(*
Nazwa:			P01_BottleFeeder
Opis:			Stacja podajnika nasadek
Wersja:			v0.1
Data:			2018-10-10
Autor:			DP
Urzadzenia:		
Konfiguracja:	
Info:

*)
PROGRAM P01_BottleFeeder
VAR_INPUT
	IbBottleFeederGate1Sensor					:BOOL;			// Czujnik otwarcia 1 szlabanu 
	IbBottleFeederGate2Sensor					:BOOL;			// Czujnik otwarcia 2 szlabanu 
	IbBottleFeederArmLeftSensor					:BOOL;			// Czujnik położenia siłownika poziomego ramienia - lewy
	IbBottleFeederArmRightSensor				:BOOL;			// Czujnik położenia siłownika poziomego ramienia - prawy
	IbBottleFeederArmUpSensor					:BOOL;			// Czujnik położenia siłownika pionowego ramienia - góra
	IbBottleFeederArmDownSensor					:BOOL;			// Czujnik polożenia siłowniak pionowego ramienia - dół
	IbBottleFeederFormPositioningClosedSensor	:BOOL;			// Czujnik schowania siłownika pozycjonujacego formatke
	IbBottleFeederBottleSensor					:BOOL;			// Czujnik obecności butelki pomiedzy szlabanami
	IbBottleFeederFormGateBeforeSensor 			:BOOL;			// Czujnik przed szlabanem formatek
	IbBottleFeederFormGateAfterSensor 			:BOOL;			// Czujnik za szlabanem formatek
	IbBottleFeederLevelSensor					:BOOL;			// Czujnik kolejki butelki
	IbBottleFeederNotInsertedSensor				AT %I*: BOOL; 	// Czujnik źle włozonej butelki za stacją	
	
END_VAR

VAR
	tonSimu1	:	TON;
	tonSimu2	:	TON;	
	tonSimu3	:	TON;	

	fbBottleFeeder						  	: FB_BottleFeeder;		// Bloczek do obsługi stacji podajnika butelek
	fbTurnTable								: FB_MitsubishiInverter; 	//Bloczek do obsługi falownika stołu obrotewego
	
	eBottleFeederStationState				: E_Station;
	eBottleFeederRunningState				: E_BottleFeederState;
	fbBottleFeederState						: FB_State;
	
	eBottleFeederTurnTableState				: E_Station;
	eBottleFeederTurnTableRunningState		: E_ConveyorState;
	fbBottleSorterTurnTableState			: FB_State;
	
	fbGateBottleFeeder						: FB_SpringGateV2;
	
	//Wyjścia sterujące
	QbBottleFeederGate1						:BOOL;			// Szlaban 1 (lewy)
	QbBottleFeederGate2						:BOOL;			// Szlaban 2 (prawy)
	QbBottleFeederArmLeft					:BOOL;			// Lewo
	QbBottleFeederArmDown					:BOOL;			// Dół
	QbBottleFeederGripper					:BOOL;			// Chwytak
	QbBottleFeederFormPositioning			:BOOL;			// Pozycjonowanie formatki
	QbBottleFeederFormGate					:BOOL;			// Szlaban formatki
	
	// Stół obrotowy
	uiBottleFeederTurnTableSW					AT %I*: UINT;
	uiBottleFeederTurnTableActualVelocity		AT %I*: UDINT;
	uiBottleFeederTurnTableCW  					AT %Q*: UINT;
	udiBottleFeederTurnTableVelocity			AT %Q*: UDINT;
	bGateRun: BOOL;
	iTest2: INT;
	bTestTurnTableRun: BOOL;
	
	bTest: BOOL;
	tonNotQbBottleFeederArmDown: TON;
END_VAR

aWarning();
aBottleFeeder();
aTurntable();
aGateTime();
aGate();

tonNotQbBottleFeederArmDown(IN:= NOT QbBottleFeederArmDown, PT:=T#50MS);


VIS.nBottleFeederTurnTableVelocityCV := uiBottleFeederTurnTableActualVelocity;

IF fbBottleFeeder.bCycleDone THEN
	bGateRun:=TRUE;
END_IF

IF fbGateBottleFeeder.bCycleDone THEN
	bGateRun:=FALSE;
END_IF

(********ASOWANIE ROZKAZÓW CYKLI*********)
IF fbBottleFeeder.bCycleDone AND bManualMode THEN
	VIS.bBottleFeederRun := FALSE;
END_IF


fbBottleFeederState(
	eState									:= eBottleFeederStationState,
	bRun									:= VIS.bBottleFeederRun,
	eBottleSorterRunningState				:= eBottleFeederRunningState,
	sStateDesc								=> VIS.sBottleFeederState,
	iState									=> VIS.iBottleFeederState);
	
(*
// tutaj dorobić obsługe wizki dla stoli obrotowego
eBottleSorterTurnTableRunningState:=eBottleSorterTurnTableState;


fbBottleSorterTurnTableState(
	eState													:= eBottleSorterTurnTableState , 
	bRun													:= GVL.bBottleSorterTurnTableRun,	
	eBottleSorterRunningState									:= eBottleSorterTurnTableRunningState , 
	sStateDesc												=> VIS.sBottleSorterTurnTableState,
	iState													=> VIS.iBottleSorterTurnTableState	);
*)

ACTION aBottleFeeder:
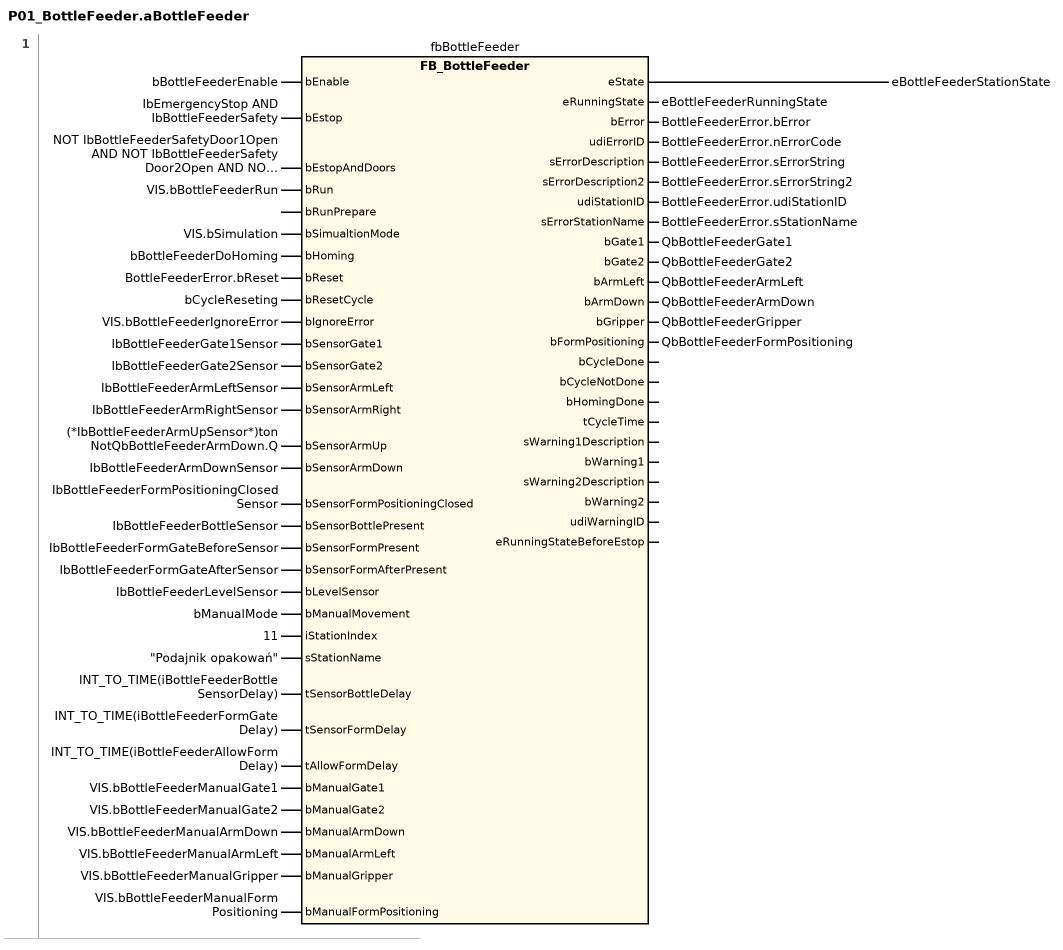
// NETWORK 1
fbBottleFeeder(
    bEnable := bBottleFeederEnable,
    bEstop := IbEmergencyStop AND IbBottleFeederSafety,
    bEstopAndDoors := NOT IbBottleFeederSafetyDoor1Open AND NOT IbBottleFeederSafetyDoor2Open AND NOT IbBottleFeederSafetyDoor3Open,
    bRun := VIS.bBottleFeederRun,
    bSimualtionMode := VIS.bSimulation,
    bHoming := bBottleFeederDoHoming,
    bReset := BottleFeederError.bReset,
    bResetCycle := bCycleReseting,
    bIgnoreError := VIS.bBottleFeederIgnoreError,
    bSensorGate1 := IbBottleFeederGate1Sensor,
    bSensorGate2 := IbBottleFeederGate2Sensor,
    bSensorArmLeft := IbBottleFeederArmLeftSensor,
    bSensorArmRight := IbBottleFeederArmRightSensor,
    bSensorArmUp := (*IbBottleFeederArmUpSensor*)tonNotQbBottleFeederArmDown.Q,
    bSensorArmDown := IbBottleFeederArmDownSensor,
    bSensorFormPositioningClosed := IbBottleFeederFormPositioningClosedSensor,
    bSensorBottlePresent := IbBottleFeederBottleSensor,
    bSensorFormPresent := IbBottleFeederFormGateBeforeSensor,
    bSensorFormAfterPresent := IbBottleFeederFormGateAfterSensor,
    bLevelSensor := IbBottleFeederLevelSensor,
    bManualMovement := bManualMode,
    iStationIndex := 11,
    sStationName := "Podajnik opakowań",
    tSensorBottleDelay := INT_TO_TIME(iBottleFeederBottleSensorDelay),
    tSensorFormDelay := INT_TO_TIME(iBottleFeederFormGateDelay),
    tAllowFormDelay := INT_TO_TIME(iBottleFeederAllowFormDelay),
    bManualGate1 := VIS.bBottleFeederManualGate1,
    bManualGate2 := VIS.bBottleFeederManualGate2,
    bManualArmDown := VIS.bBottleFeederManualArmDown,
    bManualArmLeft := VIS.bBottleFeederManualArmLeft,
    bManualGripper := VIS.bBottleFeederManualGripper,
    bManualFormPositioning := VIS.bBottleFeederManualFormPositioning,
    eRunningState => eBottleFeederRunningState,
    bError => BottleFeederError.bError,
    udiErrorID => BottleFeederError.nErrorCode,
    sErrorDescription => BottleFeederError.sErrorString,
    sErrorDescription2 => BottleFeederError.sErrorString2,
    udiStationID => BottleFeederError.udiStationID,
    sErrorStationName => BottleFeederError.sStationName,
    bGate1 => QbBottleFeederGate1,
    bGate2 => QbBottleFeederGate2,
    bArmLeft => QbBottleFeederArmLeft,
    bArmDown => QbBottleFeederArmDown,
    bGripper => QbBottleFeederGripper,
    bFormPositioning => QbBottleFeederFormPositioning); // FB_BottleFeeder
eBottleFeederStationState := fbBottleFeeder.eState;
END_ACTION

ACTION aGate:
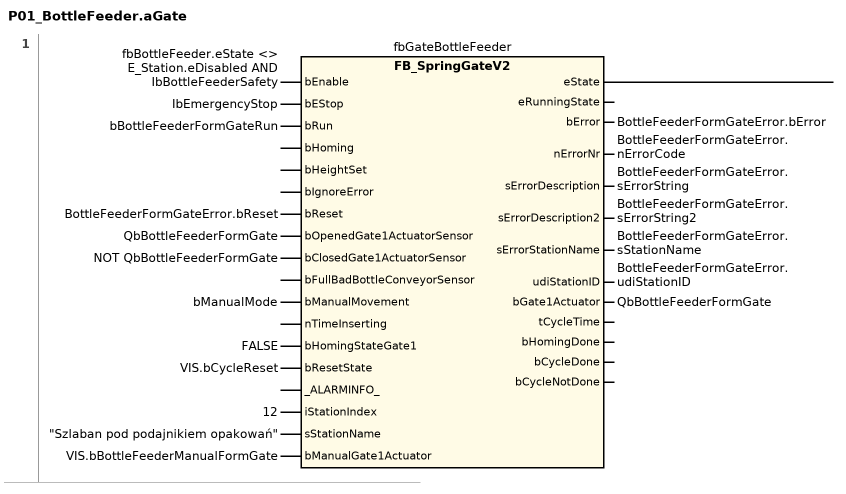
// NETWORK 1
fbGateBottleFeeder(
    bEnable := fbBottleFeeder.eState <> E_Station.eDisabled AND IbBottleFeederSafety,
    bEStop := IbEmergencyStop,
    bRun := bBottleFeederFormGateRun,
    bReset := BottleFeederFormGateError.bReset,
    bOpenedGate1ActuatorSensor := QbBottleFeederFormGate,
    bClosedGate1ActuatorSensor := NOT QbBottleFeederFormGate,
    bManualMovement := bManualMode,
    bHomingStateGate1 := FALSE,
    bResetState := VIS.bCycleReset,
    iStationIndex := 12,
    sStationName := "Szlaban pod podajnikiem opakowań",
    bManualGate1Actuator := VIS.bBottleFeederManualFormGate,
    bError => BottleFeederFormGateError.bError,
    nErrorNr => BottleFeederFormGateError.nErrorCode,
    sErrorDescription => BottleFeederFormGateError.sErrorString,
    sErrorDescription2 => BottleFeederFormGateError.sErrorString2,
    sErrorStationName => BottleFeederFormGateError.sStationName,
    udiStationID => BottleFeederFormGateError.udiStationID,
    bGate1Actuator => QbBottleFeederFormGate); // FB_SpringGateV2
END_ACTION

ACTION aGateTime:
IF bFormTransportersDispencerSlowSpeed THEN 
	fbGateBottleFeeder.nTimeInserting	:=	500;
ELSE
	fbGateBottleFeeder.nTimeInserting	:=	200;	//200
END_IF
END_ACTION

ACTION aTurntable:
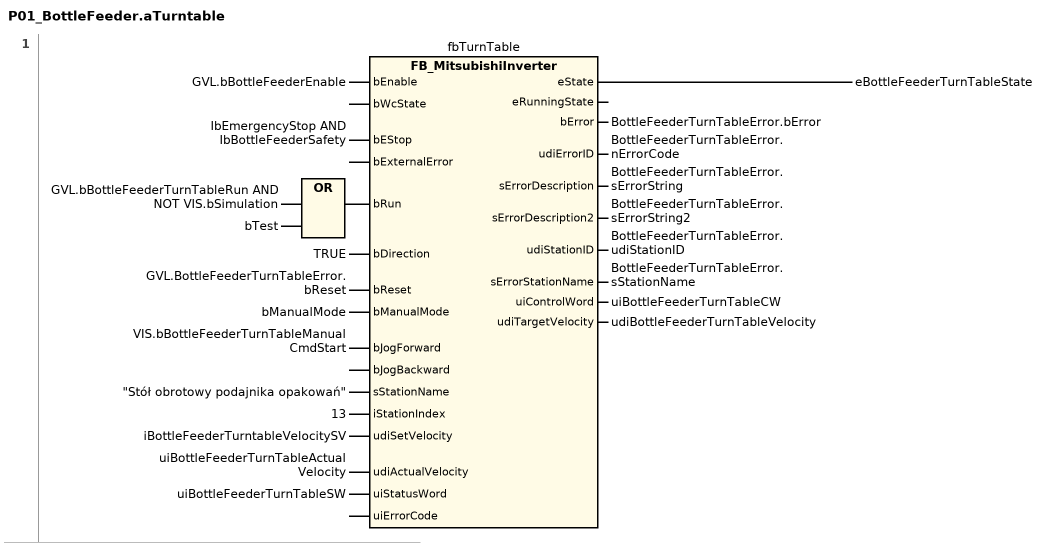
// NETWORK 1
fbTurnTable(
    bEnable := GVL.bBottleFeederEnable,
    bEStop := IbEmergencyStop AND IbBottleFeederSafety,
    bRun := (GVL.bBottleFeederTurnTableRun AND NOT VIS.bSimulation) OR bTest,
    bDirection := TRUE,
    bReset := GVL.BottleFeederTurnTableError.bReset,
    bManualMode := bManualMode,
    bJogForward := VIS.bBottleFeederTurnTableManualCmdStart,
    sStationName := "Stół obrotowy podajnika opakowań",
    iStationIndex := 13,
    udiSetVelocity := iBottleFeederTurntableVelocitySV,
    udiActualVelocity := uiBottleFeederTurnTableActualVelocity,
    uiStatusWord := uiBottleFeederTurnTableSW,
    bError => BottleFeederTurnTableError.bError,
    udiErrorID => BottleFeederTurnTableError.nErrorCode,
    sErrorDescription => BottleFeederTurnTableError.sErrorString,
    sErrorDescription2 => BottleFeederTurnTableError.sErrorString2,
    udiStationID => BottleFeederTurnTableError.udiStationID,
    sErrorStationName => BottleFeederTurnTableError.sStationName,
    uiControlWord => uiBottleFeederTurnTableCW,
    udiTargetVelocity => udiBottleFeederTurnTableVelocity); // FB_MitsubishiInverter
eBottleFeederTurnTableState := fbTurnTable.eState;
END_ACTION

ACTION aWarning:
// Warning 1
IF (IbBottleFeederSafetyDoor3Open AND bBottleFeederEnable) AND NOT BottleFeederWarning[0].bWarning THEN
	BottleFeederWarning[0].bWarning										:=TRUE;
	BottleFeederWarning[0].udiWarningCode								:=1;
	BottleFeederWarning[0].sDescription									:='Podajnik butelek | Otwarte drzwi dostępowe';
ELSIF (NOT GVL_io.IbBottleFeederSafetyDoor3Open OR NOT bBottleFeederEnable) (*AND BottleFeederWarning[0].bAcknowledge*) THEN
	BottleFeederWarning[0].bWarning										:= FALSE;
	BottleFeederWarning[0].bAcknowledge									:= FALSE;
	VIS.uliWarningAcknowledge.23 										:= FALSE;
//ELSIF BottleFeederWarning[0].bAcknowledge THEN
//ELSE
//	BottleFeederWarning[0].bAcknowledge									:= TRUE;
END_IF	

(*// Warning 2
IF (fbBottleFeeder.bWarning1 AND bBottleFeederEnable) AND NOT BottleFeederWarning[1].bWarning THEN
	BottleFeederWarning[1].bWarning										:= TRUE;
	BottleFeederWarning[1].udiWarningCode								:= 2;
	BottleFeederWarning[1].sDescription									:= 'Podajnik butelek | Niski poziom butelek';
ELSIF (NOT fbBottleFeeder.bWarning1 OR NOT bBottleFeederEnable) AND BottleFeederWarning[1].bAcknowledge THEN
	BottleFeederWarning[1].bWarning										:= FALSE;
	BottleFeederWarning[1].bAcknowledge									:= FALSE;
	VIS.uliWarningAcknowledge.26 										:= FALSE;
ELSIF BottleFeederWarning[1].bAcknowledge THEN
	BottleFeederWarning[1].bAcknowledge									:= TRUE;
END_IF*)

//Warning 3
IF (IbBottleFeederSafetyDoor1Open AND bBottleFeederEnable) AND NOT BottleFeederWarning[2].bWarning THEN
	BottleFeederWarning[2].bWarning										:=TRUE;
	BottleFeederWarning[2].udiWarningCode								:=3;
	BottleFeederWarning[2].sDescription									:='Podajnik butelek | Otwarta bramka wjazdowa';
ELSIF (NOT IbBottleFeederSafetyDoor1Open OR NOT bBottleFeederEnable) (*AND BottleFeederWarning[2].bAcknowledge*) THEN
	BottleFeederWarning[2].bWarning										:= FALSE;
	BottleFeederWarning[2].bAcknowledge									:= FALSE;
	VIS.uliWarningAcknowledge.41 										:= FALSE;
//ELSIF BottleFeederWarning[2].bAcknowledge THEN
//	BottleFeederWarning[2].bAcknowledge									:= TRUE;
END_IF	

//Warning 4
BottleFeederWarning[3].sDescription										:='Podajnik butelek | Otwarta bramka wyjazdowa';
IF (IbBottleFeederSafetyDoor2Open AND bBottleFeederEnable) AND NOT BottleFeederWarning[3].bWarning THEN
	BottleFeederWarning[3].bWarning										:=TRUE;
	BottleFeederWarning[3].udiWarningCode								:=4;
	BottleFeederWarning[3].sDescription									:='Podajnik butelek | Otwarta bramka wyjazdowa';
ELSIF (NOT GVL_io.IbBottleFeederSafetyDoor2Open OR NOT bBottleFeederEnable) (*AND BottleFeederWarning[3].bAcknowledge*) THEN
	BottleFeederWarning[3].bWarning										:= FALSE;
	BottleFeederWarning[3].bAcknowledge									:= FALSE;
	VIS.uliWarningAcknowledge.42 										:= FALSE;
//ELSIF BottleFeederWarning[3].bAcknowledge THEN
//	BottleFeederWarning[3].bAcknowledge									:= TRUE;
END_IF
END_ACTION

END_PROGRAM

(* stored: Version 1.1.0.1, ProductVersion 3.1.4026.13, FileIdentifier 157e88ac4ae68c99e4f05e3faf8bc542febd6fd0, FileSignature 503133d8b1969cb58465758c7ced616eff591c1f8869ac7c2e5f2998a2294020808ae8da15fc46838cf6bed5be8623240aac7f70421a3540d871ef445d8fbcebe5c554234cc009f9142cda6d90d6c32b0e2eb1e407ca83dc66f565005e4dd37a24b64ade721756d3de6d83a2c018fd1b144e9456b2e02030905a6531b5528db05edf17bff0184bbdabffce4c592061490d57a986bd14be13a74626e2994df37dc14c6092f0750be5805f4516d90ab757506e44ffaae45f9b6cc14c23eed39c60c95b53f05cd8f1a36a92f41c3ba28141b858fd4e8e51890c31ca526ffe85d5ca56b7adf4db616e2c4a63fe8bc271dd0060d9d8ecffd7a859db14e29f72b8ae18
   POU P01_BottleFeeder: Id {f0da2a36-64e5-4ba5-b4d6-b01f2d01a6ba}, SpecialFunc None
   Action aBottleFeeder: Id {e6d7c750-482e-4788-ab02-bb4c961a751c}
   Action aGate: Id {fd91c10a-3466-4c6f-b963-da479335c4cc}
   Action aGateTime: Id {f4aea3fc-415c-4e5a-95a5-9634a7556c2b}
   Action aTurntable: Id {eb9f3989-10af-4d30-8c7b-1ab9d18655fe}
   Action aWarning: Id {effdaae0-f15e-49fa-84fd-71c32f27af84} *)
